// TIA Portal V18 export
// export: Created 2026-01-09T11:23:40.9712194Z, ExportSetting WithDefaults, DisplayName Totally Integrated Automation Portal, DisplayVersion V18 Update 5, DisplayName TIA Portal Openness, DisplayVersion V18 Update 5, DisplayName TIA Portal Teamcenter Gateway, DisplayVersion V18, DisplayName TIA Portal Version Control Interface, DisplayVersion V18, DisplayName SINAMICS Startdrive Advanced, DisplayVersion V18 SP2 Update 1, DisplayName SINAMICS Startdrive G110M, G120, G120C, G120D, G120P, G115D, DisplayVersion V18 SP2 Update 1, DisplayName SINAMICS Startdrive G130, G150, S120, S150, SINAMICS MV, S210, G220, S200, DisplayVersion V18 SP2 Update 1, DisplayName STEP 7 Professional, DisplayVersion V18 Update 5, DisplayName STEP 7 Safety, DisplayVersion V18, DisplayName WinCC Professional, DisplayVersion V18 Update 5
Screen "630 IO Main"  1280x800, Number=630, Template=06Diagnosis
  ScreenLayer "Layer_0"
    Button "按钮_39" at 526,292 size 234x83  Mode=Text, StyleItem=BtnNormal20, TextOff="数字量输出 Q / Select Q / Vyberte Q"
      on Click: ActivateScreen(Screen name := 633 Select_Q, Object number := 0); SetTag(Tag := Sys_VersionManagement_HMIPageID, Value := 633)
    Button "按钮_40" at 283,292 size 234x83  Mode=Text, StyleItem=BtnNormal20, TextOff="数字量输入 I / Select I / Vyberte I"
      on Click: ActivateScreen(Screen name := 631Select_I, Object number := 0); SetTag(Tag := Sys_VersionManagement_HMIPageID, Value := 631)
    Button "按钮_1" at 526,397 size 234x83  Mode=Text, StyleItem=BtnNormal20, TextOff="模拟量输出 PQW / Analog Output / Analógový výstup", TextOn="模拟量输出 PQW / Analog Output / Analógový výstup"
      on Click: ActivateScreen(Screen name := 636 Analog Output, Object number := 0); SetTag(Tag := Sys_VersionManagement_HMIPageID, Value := 636)
    Button "按钮_2" at 283,397 size 234x83  Mode=Text, StyleItem=BtnNormal20, TextOff="模拟量输入 PIW / Analog Input / Analógový vstup", TextOn="模拟量输入 PIW / Analog Input / Analógový vstup"
      on Click: ActivateScreen(Screen name := 635 Analog Input, Object number := 0); SetTag(Tag := Sys_VersionManagement_HMIPageID, Value := 635)
